// TIA Portal V17 export
// export: Created 2024-09-02T12:50:26.5651958Z, ExportSetting WithDefaults, DisplayName Totally Integrated Automation Portal, DisplayVersion V17, DisplayName TIA Portal Openness, DisplayVersion V17, DisplayName TIA Portal Version Control Interface, DisplayVersion V17, DisplayName STEP 7 Professional, DisplayVersion V17, DisplayName STEP 7 Safety, DisplayVersion V17, DisplayName WinCC Professional, DisplayVersion V17
TYPE "TypeTypeChange"
// stored: IsFailsafeCompliant false
   STRUCT
      Start : Bool;   // Start Auswertung / Start evaluation
      Quit : Bool;   // Typwechsel Quittieren / Acknowledge type change
      Reset : Bool;   // Speicher loeschen / Clear memory
      TypeChange : Bool;   // Typwechsel steht an / Type change pending
      no_TypeChange : Bool;   // kein Typwechsel / no type change
      Error_Parameter : Bool;   // Fehler Parameter / Error Parameter
      Data : Array[1..64] of Byte;   // aktuelle Daten / Current Data
      Memory : Array[1..64] of Byte;   // Speicher / Memory
      HM : Array[1..8] of Bool;
   END_STRUCT;
END_TYPE
